// TIA Portal V16 export
// export: Created 2021-11-12T13:33:10.1366226Z, ExportSetting WithDefaults, DisplayName Totally Integrated Automation Portal, DisplayVersion V16 Update 3, DisplayName TIA Portal Version Control Interface, DisplayVersion V16 Update 2, DisplayName TIA Portal Openness, DisplayVersion V16 Update 3, DisplayName SINAMICS Startdrive Advanced, DisplayVersion V16 Update 5, DisplayName SINAMICS Startdrive G130, G150, S120, S150, SINAMICS MV, S210, DisplayVersion V16 Update 5, DisplayName SINAMICS Startdrive G110M, G120, G120C, G120D, G120P, G115D, DisplayVersion V16 Update 5, DisplayName STEP 7 Professional, DisplayVersion V16 Update 3, DisplayName STEP 7 Safety, DisplayVersion V16, DisplayName WinCC UA Professional, DisplayVersion V16 Update 3
FUNCTION_BLOCK "Station450"   // FB58, LAD
{ S7_Optimized_Access := 'TRUE' }
VERSION : 0.1
// stored: AutoNumber true, IsIECCheckEnabled false, IsRetainMemResEnabled false, MemoryReserve 100, SetENOAutomatically false, UDAEnableTagReadback false
   VAR
      SF_GL01_MA01 : "STD_Drive1";
      SF_GL02_MA01 { S7_SetPoint := 'True'} : "STD_Drive1";
      SF_GL03_MA01 { S7_SetPoint := 'True'} : "STD_Drive1";
      SF_GL04_MA01 { S7_SetPoint := 'True'} : "STD_Drive1";
      SF_UC21_TA1 { S7_SetPoint := 'True'} : "STD_Siemens_G120_CU240E_2_PN";
      SF_UC21_TA2 { S7_SetPoint := 'True'} : "STD_Siemens_G120_CU240E_2_PN";
      SF_UC21_TA3 { S7_SetPoint := 'True'} : "STD_Siemens_G120_CU240E_2_PN";
      SF_UC21_TA4 { S7_SetPoint := 'True'} : "STD_Siemens_G120_CU240E_2_PN";
      SF_BoxPartCounter { S7_SetPoint := 'True'} : "STD_PartCounter";
      SF_TON_BOX { S7_SetPoint := 'True'} : TON_TIME;
      SF_TOF_430TA01 { S7_SetPoint := 'True'} : TOF_TIME;   // TOF timer to stop conv after 430TA01 stopped
      SF_TOF_450TA01 { S7_SetPoint := 'True'} : TOF_TIME;   // TOF timer to stop conv after 450TA01 stopped
      SF_TOF_450TA02_1 { S7_SetPoint := 'True'} : TOF_TIME;   // TOF timer to stop conv after 450TA02 stopped
      SF_TOF_450TA02_2 { S7_SetPoint := 'True'} : TOF_TIME;   // TOF timer to stop conv after 450TA02 stopped
      SF_TOF_450TA04 { S7_SetPoint := 'True'} : TOF_TIME;   // TOF timer to stop conv after 450TA03 stopped
      SB1_PowerOk { S7_SetPoint := 'True'} : Bool;
      SB1BoxExchangeReq : Bool;   // Box - exchange request
      SF_CL01_Alarm { S7_SetPoint := 'True'} : "STD_DI_Mon";
      SF_CL01_Warning { S7_SetPoint := 'True'} : "STD_DI_Mon";
   END_VAR
   VAR_TEMP
      TS_GL01MA01 : "UDT_DriveControl";
      TS_GL02MA01 : "UDT_DriveControl";
      TS_GL03MA01 : "UDT_DriveControl";
      TS_GL04MA01 : "UDT_DriveControl";
      TS_UC21TA01 : Struct
         ReqDir1 : Bool;   // Move in direction 1
         ReqDir2 : Bool;   // Move in direction 2
         AckErr : Bool;   // Acknowledge error
         SpeedSP : Real;   // Speed setpoint
      END_STRUCT;
      TS_UC21TA02 : Struct
         ReqDir1 : Bool;   // Move in direction 1
         ReqDir2 : Bool;   // Move in direction 2
         AckErr : Bool;   // Acknowledge error
         SpeedSP : Real;   // Speed setpoint
      END_STRUCT;
      TS_UC21TA03 : Struct
         ReqDir1 : Bool;   // Move in direction 1
         ReqDir2 : Bool;   // Move in direction 2
         AckErr : Bool;   // Acknowledge error
         SpeedSP : Real;   // Speed setpoint
      END_STRUCT;
      TS_UC21TA04 : Struct
         ReqDir1 : Bool;   // Move in direction 1
         ReqDir2 : Bool;   // Move in direction 2
         AckErr : Bool;   // Acknowledge error
         SpeedSP : Real;   // Speed setpoint
      END_STRUCT;
      TI_NoOfParts : Int;   // Number of parts per one pulse
      TB1BoxFull : Bool;   // Box is full
   END_VAR
BEGIN

REGION Network 1: ***************ClearTemporary***************
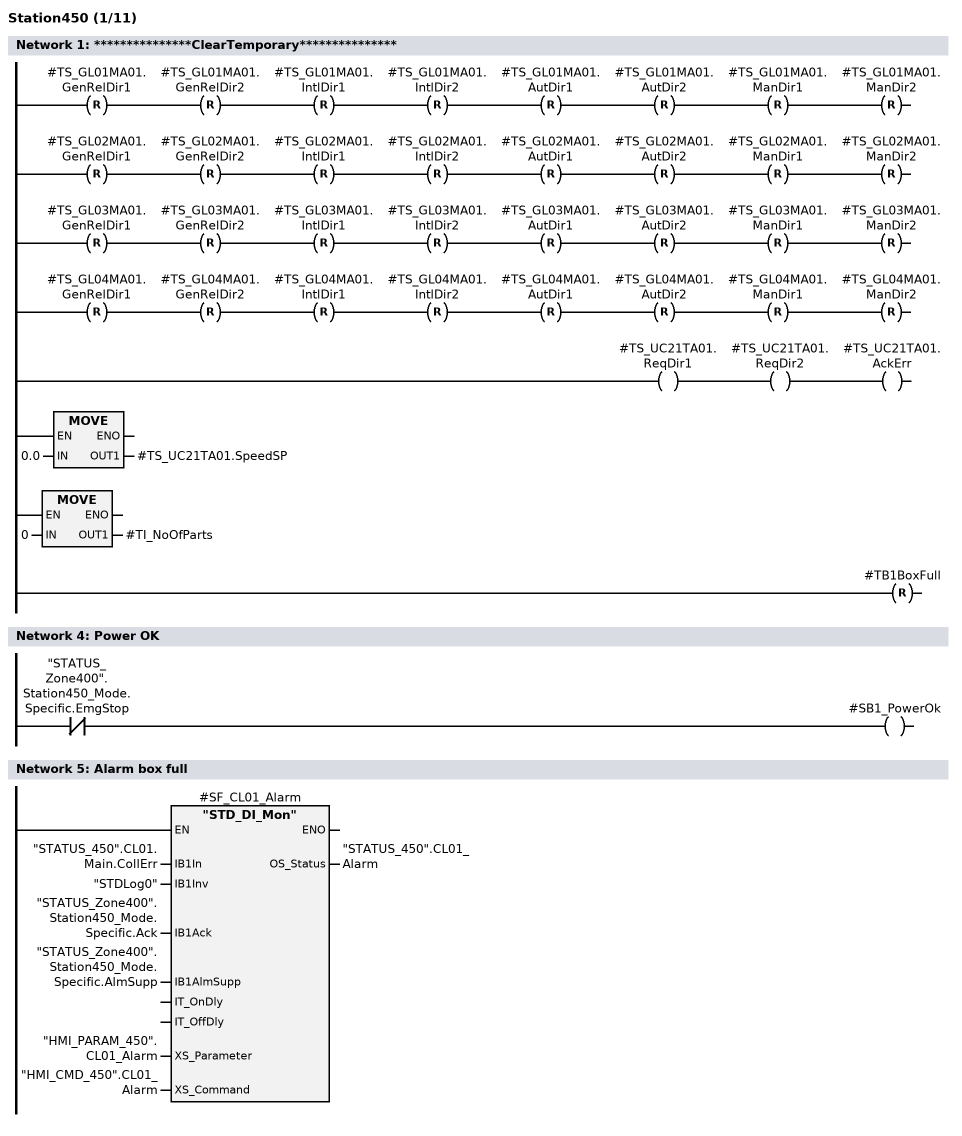
   RUNG wire#powerrail
      R_Coil( #TS_GL01MA01.GenRelDir1 )
      R_Coil( #TS_GL01MA01.GenRelDir2 )
      R_Coil( #TS_GL01MA01.IntlDir1 )
      R_Coil( #TS_GL01MA01.IntlDir2 )
      R_Coil( #TS_GL01MA01.AutDir1 )
      R_Coil( #TS_GL01MA01.AutDir2 )
      R_Coil( #TS_GL01MA01.ManDir1 )
      R_Coil( #TS_GL01MA01.ManDir2 )
   END_RUNG
   RUNG wire#powerrail
      R_Coil( #TS_GL02MA01.GenRelDir1 )
      R_Coil( #TS_GL02MA01.GenRelDir2 )
      R_Coil( #TS_GL02MA01.IntlDir1 )
      R_Coil( #TS_GL02MA01.IntlDir2 )
      R_Coil( #TS_GL02MA01.AutDir1 )
      R_Coil( #TS_GL02MA01.AutDir2 )
      R_Coil( #TS_GL02MA01.ManDir1 )
      R_Coil( #TS_GL02MA01.ManDir2 )
   END_RUNG
   RUNG wire#powerrail
      R_Coil( #TS_GL03MA01.GenRelDir1 )
      R_Coil( #TS_GL03MA01.GenRelDir2 )
      R_Coil( #TS_GL03MA01.IntlDir1 )
      R_Coil( #TS_GL03MA01.IntlDir2 )
      R_Coil( #TS_GL03MA01.AutDir1 )
      R_Coil( #TS_GL03MA01.AutDir2 )
      R_Coil( #TS_GL03MA01.ManDir1 )
      R_Coil( #TS_GL03MA01.ManDir2 )
   END_RUNG
   RUNG wire#powerrail
      R_Coil( #TS_GL04MA01.GenRelDir1 )
      R_Coil( #TS_GL04MA01.GenRelDir2 )
      R_Coil( #TS_GL04MA01.IntlDir1 )
      R_Coil( #TS_GL04MA01.IntlDir2 )
      R_Coil( #TS_GL04MA01.AutDir1 )
      R_Coil( #TS_GL04MA01.AutDir2 )
      R_Coil( #TS_GL04MA01.ManDir1 )
      R_Coil( #TS_GL04MA01.ManDir2 )
   END_RUNG
   RUNG wire#powerrail
      Coil( #TS_UC21TA01.ReqDir1 )
      Coil( #TS_UC21TA01.ReqDir2 )
      Coil( #TS_UC21TA01.AckErr )
   END_RUNG
   RUNG wire#powerrail
      Move(in := 0.0, out1 => #TS_UC21TA01.SpeedSP)
   END_RUNG
   RUNG wire#powerrail
      Move(in := 0, out1 => #TI_NoOfParts)
   END_RUNG
   RUNG wire#powerrail
      R_Coil( #TB1BoxFull )
   END_RUNG
   // the same network as SCL:
   #TS_GL01MA01.GenRelDir1 := FALSE;
   #TS_GL01MA01.GenRelDir2 := FALSE;
   #TS_GL01MA01.IntlDir1 := FALSE;
   #TS_GL01MA01.IntlDir2 := FALSE;
   #TS_GL01MA01.AutDir1 := FALSE;
   #TS_GL01MA01.AutDir2 := FALSE;
   #TS_GL01MA01.ManDir1 := FALSE;
   #TS_GL01MA01.ManDir2 := FALSE;
   #TS_GL02MA01.GenRelDir1 := FALSE;
   #TS_GL02MA01.GenRelDir2 := FALSE;
   #TS_GL02MA01.IntlDir1 := FALSE;
   #TS_GL02MA01.IntlDir2 := FALSE;
   #TS_GL02MA01.AutDir1 := FALSE;
   #TS_GL02MA01.AutDir2 := FALSE;
   #TS_GL02MA01.ManDir1 := FALSE;
   #TS_GL02MA01.ManDir2 := FALSE;
   #TS_GL03MA01.GenRelDir1 := FALSE;
   #TS_GL03MA01.GenRelDir2 := FALSE;
   #TS_GL03MA01.IntlDir1 := FALSE;
   #TS_GL03MA01.IntlDir2 := FALSE;
   #TS_GL03MA01.AutDir1 := FALSE;
   #TS_GL03MA01.AutDir2 := FALSE;
   #TS_GL03MA01.ManDir1 := FALSE;
   #TS_GL03MA01.ManDir2 := FALSE;
   #TS_GL04MA01.GenRelDir1 := FALSE;
   #TS_GL04MA01.GenRelDir2 := FALSE;
   #TS_GL04MA01.IntlDir1 := FALSE;
   #TS_GL04MA01.IntlDir2 := FALSE;
   #TS_GL04MA01.AutDir1 := FALSE;
   #TS_GL04MA01.AutDir2 := FALSE;
   #TS_GL04MA01.ManDir1 := FALSE;
   #TS_GL04MA01.ManDir2 := FALSE;
   #TS_UC21TA01.ReqDir1 := TRUE;
   #TS_UC21TA01.ReqDir2 := TRUE;
   #TS_UC21TA01.AckErr := TRUE;
   #TS_UC21TA01.SpeedSP := 0.0;
   #TI_NoOfParts := 0;
   #TB1BoxFull := FALSE;
END_REGION

REGION Network 2: ***************SensorsAlarms***************
END_REGION

REGION Network 3: ***************ProcesAlarms***************
END_REGION

REGION Network 4: Power OK
   RUNG wire#powerrail
      I_Contact( "STATUS_Zone400".Station450_Mode.Specific.EmgStop )
      Coil( #SB1_PowerOk )
   END_RUNG
   // the same network as SCL:
   #SB1_PowerOk := NOT "STATUS_Zone400".Station450_Mode.Specific.EmgStop;
END_REGION

REGION Network 5: Alarm box full
   RUNG wire#powerrail
      #SF_CL01_Alarm(IB1In := "STATUS_450".CL01.Main.CollErr, IB1Inv := "STDLog0", IB1Ack := "STATUS_Zone400".Station450_Mode.Specific.Ack, IB1AlmSupp := "STATUS_Zone400".Station450_Mode.Specific.AlmSupp, IT_OnDly :=, IT_OffDly :=, XS_Parameter := "HMI_PARAM_450".CL01_Alarm, XS_Command := "HMI_CMD_450".CL01_Alarm, OS_Status => "STATUS_450".CL01_Alarm)
   END_RUNG
   // the same network as SCL:
   #SF_CL01_Alarm(IB1In := "STATUS_450".CL01.Main.CollErr,   // "STD_DI_Mon"
                  IB1Inv := "STDLog0",
                  IB1Ack := "STATUS_Zone400".Station450_Mode.Specific.Ack,
                  IB1AlmSupp := "STATUS_Zone400".Station450_Mode.Specific.AlmSupp,
                  XS_Parameter := "HMI_PARAM_450".CL01_Alarm,
                  XS_Command := "HMI_CMD_450".CL01_Alarm,
                  OS_Status => "STATUS_450".CL01_Alarm);
END_REGION

REGION Network 6: Warning box almost full
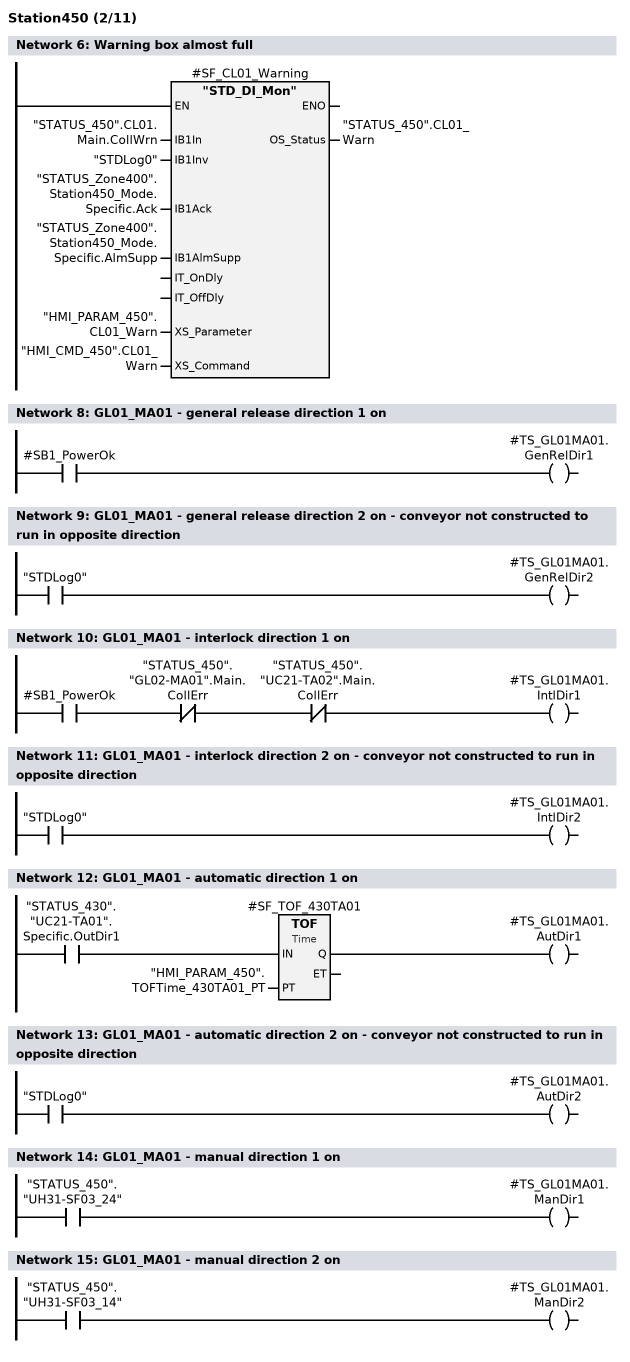
   RUNG wire#powerrail
      #SF_CL01_Warning(IB1In := "STATUS_450".CL01.Main.CollWrn, IB1Inv := "STDLog0", IB1Ack := "STATUS_Zone400".Station450_Mode.Specific.Ack, IB1AlmSupp := "STATUS_Zone400".Station450_Mode.Specific.AlmSupp, IT_OnDly :=, IT_OffDly :=, XS_Parameter := "HMI_PARAM_450".CL01_Warn, XS_Command := "HMI_CMD_450".CL01_Warn, OS_Status => "STATUS_450".CL01_Warn)
   END_RUNG
   // the same network as SCL:
   #SF_CL01_Warning(IB1In := "STATUS_450".CL01.Main.CollWrn,   // "STD_DI_Mon"
                    IB1Inv := "STDLog0",
                    IB1Ack := "STATUS_Zone400".Station450_Mode.Specific.Ack,
                    IB1AlmSupp := "STATUS_Zone400".Station450_Mode.Specific.AlmSupp,
                    XS_Parameter := "HMI_PARAM_450".CL01_Warn,
                    XS_Command := "HMI_CMD_450".CL01_Warn,
                    OS_Status => "STATUS_450".CL01_Warn);
END_REGION

REGION Network 7: ***************GL01_MA01 Conveyor M2***************
END_REGION

REGION Network 8: GL01_MA01 - general release direction 1 on
   RUNG wire#powerrail
      Contact( #SB1_PowerOk )
      Coil( #TS_GL01MA01.GenRelDir1 )
   END_RUNG
   // the same network as SCL:
   #TS_GL01MA01.GenRelDir1 := #SB1_PowerOk;
END_REGION

REGION Network 9: GL01_MA01 - general release direction 2 on - conveyor not constructed to run in opposite direction
   RUNG wire#powerrail
      Contact( "STDLog0" )
      Coil( #TS_GL01MA01.GenRelDir2 )
   END_RUNG
   // the same network as SCL:
   #TS_GL01MA01.GenRelDir2 := "STDLog0";
END_REGION

REGION Network 10: GL01_MA01 - interlock direction 1 on
   RUNG wire#powerrail
      Contact( #SB1_PowerOk )
      I_Contact( "STATUS_450"."GL02-MA01".Main.CollErr )
      I_Contact( "STATUS_450"."UC21-TA02".Main.CollErr )
      Coil( #TS_GL01MA01.IntlDir1 )
   END_RUNG
   // the same network as SCL:
   #TS_GL01MA01.IntlDir1 := #SB1_PowerOk AND NOT "STATUS_450"."GL02-MA01".Main.CollErr AND NOT "STATUS_450"."UC21-TA02".Main.CollErr;
END_REGION

REGION Network 11: GL01_MA01 - interlock direction 2 on - conveyor not constructed to run in opposite direction
   RUNG wire#powerrail
      Contact( "STDLog0" )
      Coil( #TS_GL01MA01.IntlDir2 )
   END_RUNG
   // the same network as SCL:
   #TS_GL01MA01.IntlDir2 := "STDLog0";
END_REGION

REGION Network 12: GL01_MA01 - automatic direction 1 on
   RUNG wire#powerrail
      Contact( "STATUS_430"."UC21-TA01".Specific.OutDir1 )
      { S7_Templates := "time_type := Time" } #SF_TOF_430TA01.TOF(pt := "HMI_PARAM_450".TOFTime_430TA01_PT, et =>)
      Coil( #TS_GL01MA01.AutDir1 )
   END_RUNG
   // the same network as SCL:
   #SF_TOF_430TA01(IN := "STATUS_430"."UC21-TA01".Specific.OutDir1, PT := "HMI_PARAM_450".TOFTime_430TA01_PT);   // TOF
   #TS_GL01MA01.AutDir1 := #SF_TOF_430TA01.Q;
END_REGION

REGION Network 13: GL01_MA01 - automatic direction 2 on - conveyor not constructed to run in opposite direction
   RUNG wire#powerrail
      Contact( "STDLog0" )
      Coil( #TS_GL01MA01.AutDir2 )
   END_RUNG
   // the same network as SCL:
   #TS_GL01MA01.AutDir2 := "STDLog0";
END_REGION

REGION Network 14: GL01_MA01 - manual direction 1 on
   RUNG wire#powerrail
      Contact( "STATUS_450"."UH31-SF03_24" )
      Coil( #TS_GL01MA01.ManDir1 )
   END_RUNG
   // the same network as SCL:
   #TS_GL01MA01.ManDir1 := "STATUS_450"."UH31-SF03_24";
END_REGION

REGION Network 15: GL01_MA01 - manual direction 2 on
   RUNG wire#powerrail
      Contact( "STATUS_450"."UH31-SF03_14" )
      Coil( #TS_GL01MA01.ManDir2 )
   END_RUNG
   // the same network as SCL:
   #TS_GL01MA01.ManDir2 := "STATUS_450"."UH31-SF03_14";
END_REGION

REGION Network 16: GL01_MA01 Drive block call
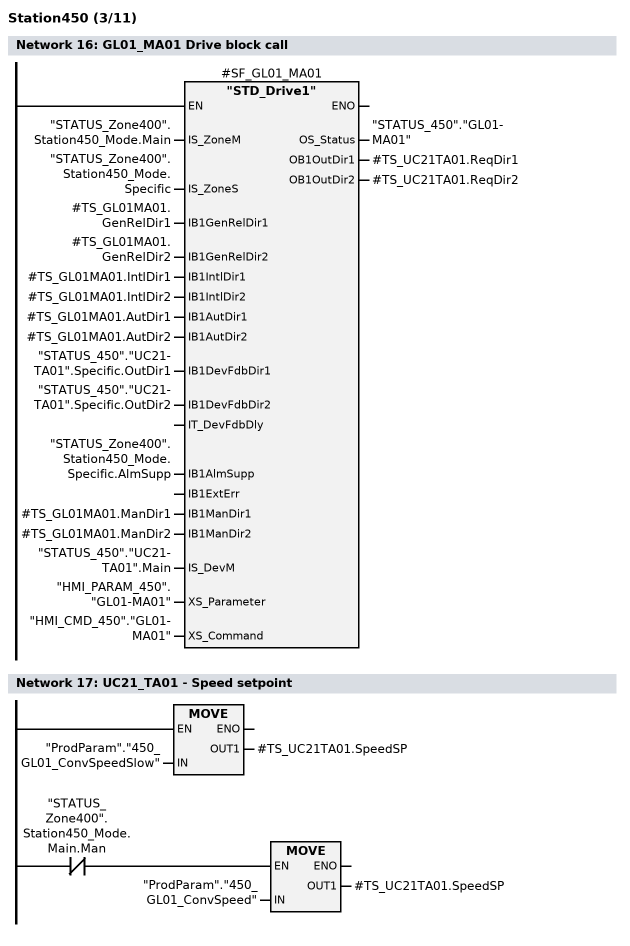
   RUNG wire#powerrail
      #SF_GL01_MA01(IS_ZoneM := "STATUS_Zone400".Station450_Mode.Main, IS_ZoneS := "STATUS_Zone400".Station450_Mode.Specific, IB1GenRelDir1 := #TS_GL01MA01.GenRelDir1, IB1GenRelDir2 := #TS_GL01MA01.GenRelDir2, IB1IntlDir1 := #TS_GL01MA01.IntlDir1, IB1IntlDir2 := #TS_GL01MA01.IntlDir2, IB1AutDir1 := #TS_GL01MA01.AutDir1, IB1AutDir2 := #TS_GL01MA01.AutDir2, IB1DevFdbDir1 := "STATUS_450"."UC21-TA01".Specific.OutDir1, IB1DevFdbDir2 := "STATUS_450"."UC21-TA01".Specific.OutDir2, IT_DevFdbDly :=, IB1AlmSupp := "STATUS_Zone400".Station450_Mode.Specific.AlmSupp, IB1ExtErr :=, IB1ManDir1 := #TS_GL01MA01.ManDir1, IB1ManDir2 := #TS_GL01MA01.ManDir2, IS_DevM := "STATUS_450"."UC21-TA01".Main, XS_Parameter := "HMI_PARAM_450"."GL01-MA01", XS_Command := "HMI_CMD_450"."GL01-MA01", OS_Status => "STATUS_450"."GL01-MA01", OB1OutDir1 => #TS_UC21TA01.ReqDir1, OB1OutDir2 => #TS_UC21TA01.ReqDir2)
   END_RUNG
   // the same network as SCL:
   #SF_GL01_MA01(IS_ZoneM := "STATUS_Zone400".Station450_Mode.Main,   // "STD_Drive1"
                 IS_ZoneS := "STATUS_Zone400".Station450_Mode.Specific,
                 IB1GenRelDir1 := #TS_GL01MA01.GenRelDir1,
                 IB1GenRelDir2 := #TS_GL01MA01.GenRelDir2,
                 IB1IntlDir1 := #TS_GL01MA01.IntlDir1,
                 IB1IntlDir2 := #TS_GL01MA01.IntlDir2,
                 IB1AutDir1 := #TS_GL01MA01.AutDir1,
                 IB1AutDir2 := #TS_GL01MA01.AutDir2,
                 IB1DevFdbDir1 := "STATUS_450"."UC21-TA01".Specific.OutDir1,
                 IB1DevFdbDir2 := "STATUS_450"."UC21-TA01".Specific.OutDir2,
                 IB1AlmSupp := "STATUS_Zone400".Station450_Mode.Specific.AlmSupp,
                 IB1ManDir1 := #TS_GL01MA01.ManDir1,
                 IB1ManDir2 := #TS_GL01MA01.ManDir2,
                 IS_DevM := "STATUS_450"."UC21-TA01".Main,
                 XS_Parameter := "HMI_PARAM_450"."GL01-MA01",
                 XS_Command := "HMI_CMD_450"."GL01-MA01",
                 OS_Status => "STATUS_450"."GL01-MA01",
                 OB1OutDir1 => #TS_UC21TA01.ReqDir1,
                 OB1OutDir2 => #TS_UC21TA01.ReqDir2);
END_REGION

REGION Network 17: UC21_TA01 - Speed setpoint
   RUNG wire#powerrail
      Move(in := "ProdParam"."450_GL01_ConvSpeedSlow", out1 => #TS_UC21TA01.SpeedSP)
   END_RUNG
   RUNG wire#powerrail
      I_Contact( "STATUS_Zone400".Station450_Mode.Main.Man )
      Move(in := "ProdParam"."450_GL01_ConvSpeed", out1 => #TS_UC21TA01.SpeedSP)
   END_RUNG
   // the same network as SCL:
   #TS_UC21TA01.SpeedSP := "ProdParam"."450_GL01_ConvSpeedSlow";
   IF NOT "STATUS_Zone400".Station450_Mode.Main.Man THEN
       #TS_UC21TA01.SpeedSP := "ProdParam"."450_GL01_ConvSpeed";
   END_IF;
END_REGION

REGION Network 18: UC21_TA01 - Frequency convertor block call
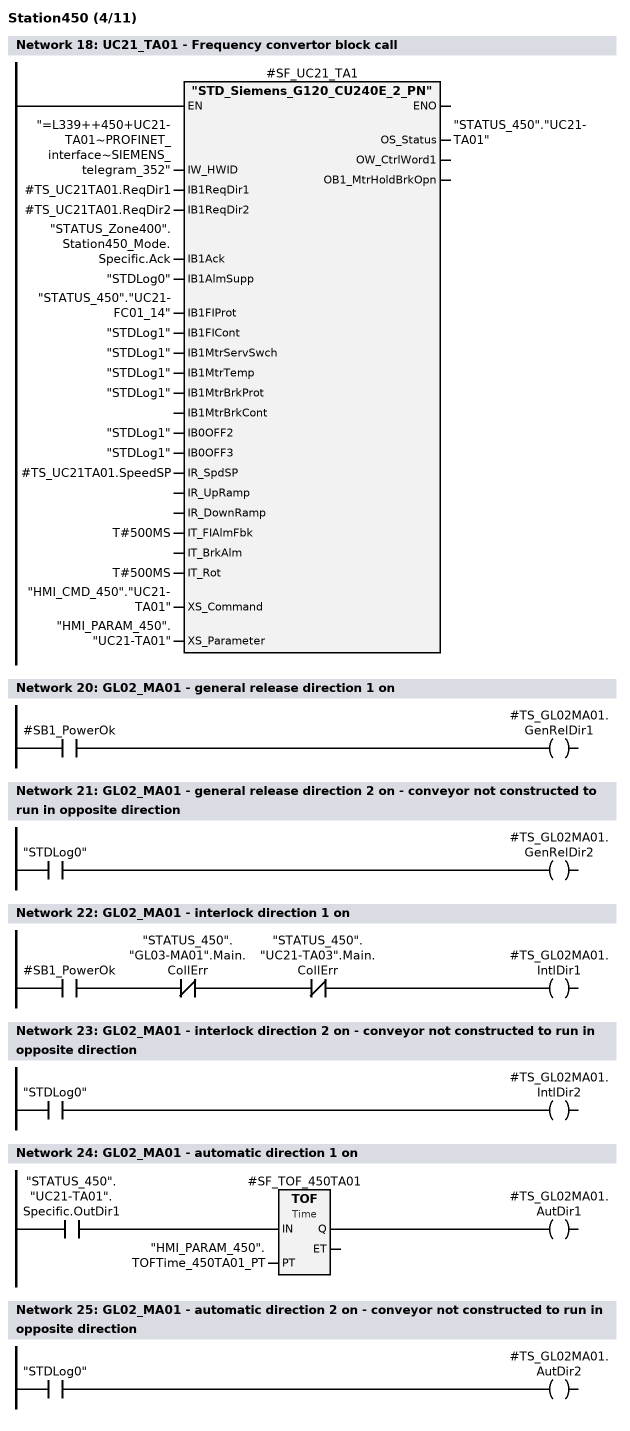
   RUNG wire#powerrail
      #SF_UC21_TA1(IW_HWID := "=L339++450+UC21-TA01~PROFINET_interface~SIEMENS_telegram_352", IB1ReqDir1 := #TS_UC21TA01.ReqDir1, IB1ReqDir2 := #TS_UC21TA01.ReqDir2, IB1Ack := "STATUS_Zone400".Station450_Mode.Specific.Ack, IB1AlmSupp := "STDLog0", IB1FIProt := "STATUS_450"."UC21-FC01_14", IB1FICont := "STDLog1", IB1MtrServSwch := "STDLog1", IB1MtrTemp := "STDLog1", IB1MtrBrkProt := "STDLog1", IB1MtrBrkCont :=, IB0OFF2 := "STDLog1", IB0OFF3 := "STDLog1", IR_SpdSP := #TS_UC21TA01.SpeedSP, IR_UpRamp :=, IR_DownRamp :=, IT_FIAlmFbk := T#500MS, IT_BrkAlm :=, IT_Rot := T#500MS, XS_Command := "HMI_CMD_450"."UC21-TA01", XS_Parameter := "HMI_PARAM_450"."UC21-TA01", OS_Status => "STATUS_450"."UC21-TA01", OW_CtrlWord1 =>, OB1_MtrHoldBrkOpn =>)
   END_RUNG
   // the same network as SCL:
   #SF_UC21_TA1(IW_HWID := "=L339++450+UC21-TA01~PROFINET_interface~SIEMENS_telegram_352",   // "STD_Siemens_G120_CU240E_2_PN"
                IB1ReqDir1 := #TS_UC21TA01.ReqDir1,
                IB1ReqDir2 := #TS_UC21TA01.ReqDir2,
                IB1Ack := "STATUS_Zone400".Station450_Mode.Specific.Ack,
                IB1AlmSupp := "STDLog0",
                IB1FIProt := "STATUS_450"."UC21-FC01_14",
                IB1FICont := "STDLog1",
                IB1MtrServSwch := "STDLog1",
                IB1MtrTemp := "STDLog1",
                IB1MtrBrkProt := "STDLog1",
                IB0OFF2 := "STDLog1",
                IB0OFF3 := "STDLog1",
                IR_SpdSP := #TS_UC21TA01.SpeedSP,
                IT_FIAlmFbk := T#500MS,
                IT_Rot := T#500MS,
                XS_Command := "HMI_CMD_450"."UC21-TA01",
                XS_Parameter := "HMI_PARAM_450"."UC21-TA01",
                OS_Status => "STATUS_450"."UC21-TA01");
END_REGION

REGION Network 19: ***************GL02_MA01 Conveyor M4***************
END_REGION

REGION Network 20: GL02_MA01 - general release direction 1 on
   RUNG wire#powerrail
      Contact( #SB1_PowerOk )
      Coil( #TS_GL02MA01.GenRelDir1 )
   END_RUNG
   // the same network as SCL:
   #TS_GL02MA01.GenRelDir1 := #SB1_PowerOk;
END_REGION

REGION Network 21: GL02_MA01 - general release direction 2 on - conveyor not constructed to run in opposite direction
   RUNG wire#powerrail
      Contact( "STDLog0" )
      Coil( #TS_GL02MA01.GenRelDir2 )
   END_RUNG
   // the same network as SCL:
   #TS_GL02MA01.GenRelDir2 := "STDLog0";
END_REGION

REGION Network 22: GL02_MA01 - interlock direction 1 on
   RUNG wire#powerrail
      Contact( #SB1_PowerOk )
      I_Contact( "STATUS_450"."GL03-MA01".Main.CollErr )
      I_Contact( "STATUS_450"."UC21-TA03".Main.CollErr )
      Coil( #TS_GL02MA01.IntlDir1 )
   END_RUNG
   // the same network as SCL:
   #TS_GL02MA01.IntlDir1 := #SB1_PowerOk AND NOT "STATUS_450"."GL03-MA01".Main.CollErr AND NOT "STATUS_450"."UC21-TA03".Main.CollErr;
END_REGION

REGION Network 23: GL02_MA01 - interlock direction 2 on - conveyor not constructed to run in opposite direction
   RUNG wire#powerrail
      Contact( "STDLog0" )
      Coil( #TS_GL02MA01.IntlDir2 )
   END_RUNG
   // the same network as SCL:
   #TS_GL02MA01.IntlDir2 := "STDLog0";
END_REGION

REGION Network 24: GL02_MA01 - automatic direction 1 on
   RUNG wire#powerrail
      Contact( "STATUS_450"."UC21-TA01".Specific.OutDir1 )
      { S7_Templates := "time_type := Time" } #SF_TOF_450TA01.TOF(pt := "HMI_PARAM_450".TOFTime_450TA01_PT, et =>)
      Coil( #TS_GL02MA01.AutDir1 )
   END_RUNG
   // the same network as SCL:
   #SF_TOF_450TA01(IN := "STATUS_450"."UC21-TA01".Specific.OutDir1, PT := "HMI_PARAM_450".TOFTime_450TA01_PT);   // TOF
   #TS_GL02MA01.AutDir1 := #SF_TOF_450TA01.Q;
END_REGION

REGION Network 25: GL02_MA01 - automatic direction 2 on - conveyor not constructed to run in opposite direction
   RUNG wire#powerrail
      Contact( "STDLog0" )
      Coil( #TS_GL02MA01.AutDir2 )
   END_RUNG
   // the same network as SCL:
   #TS_GL02MA01.AutDir2 := "STDLog0";
END_REGION

REGION Network 26: GL02_MA01 - manual direction 1 on
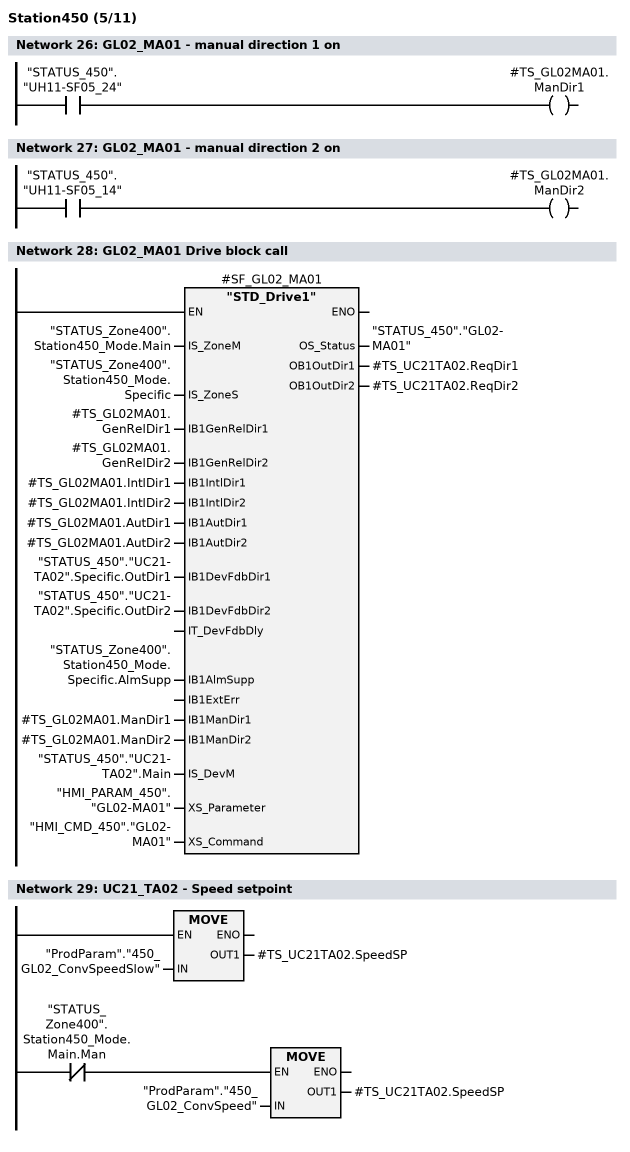
   RUNG wire#powerrail
      Contact( "STATUS_450"."UH11-SF05_24" )
      Coil( #TS_GL02MA01.ManDir1 )
   END_RUNG
   // the same network as SCL:
   #TS_GL02MA01.ManDir1 := "STATUS_450"."UH11-SF05_24";
END_REGION

REGION Network 27: GL02_MA01 - manual direction 2 on
   RUNG wire#powerrail
      Contact( "STATUS_450"."UH11-SF05_14" )
      Coil( #TS_GL02MA01.ManDir2 )
   END_RUNG
   // the same network as SCL:
   #TS_GL02MA01.ManDir2 := "STATUS_450"."UH11-SF05_14";
END_REGION

REGION Network 28: GL02_MA01 Drive block call
   RUNG wire#powerrail
      #SF_GL02_MA01(IS_ZoneM := "STATUS_Zone400".Station450_Mode.Main, IS_ZoneS := "STATUS_Zone400".Station450_Mode.Specific, IB1GenRelDir1 := #TS_GL02MA01.GenRelDir1, IB1GenRelDir2 := #TS_GL02MA01.GenRelDir2, IB1IntlDir1 := #TS_GL02MA01.IntlDir1, IB1IntlDir2 := #TS_GL02MA01.IntlDir2, IB1AutDir1 := #TS_GL02MA01.AutDir1, IB1AutDir2 := #TS_GL02MA01.AutDir2, IB1DevFdbDir1 := "STATUS_450"."UC21-TA02".Specific.OutDir1, IB1DevFdbDir2 := "STATUS_450"."UC21-TA02".Specific.OutDir2, IT_DevFdbDly :=, IB1AlmSupp := "STATUS_Zone400".Station450_Mode.Specific.AlmSupp, IB1ExtErr :=, IB1ManDir1 := #TS_GL02MA01.ManDir1, IB1ManDir2 := #TS_GL02MA01.ManDir2, IS_DevM := "STATUS_450"."UC21-TA02".Main, XS_Parameter := "HMI_PARAM_450"."GL02-MA01", XS_Command := "HMI_CMD_450"."GL02-MA01", OS_Status => "STATUS_450"."GL02-MA01", OB1OutDir1 => #TS_UC21TA02.ReqDir1, OB1OutDir2 => #TS_UC21TA02.ReqDir2)
   END_RUNG
   // the same network as SCL:
   #SF_GL02_MA01(IS_ZoneM := "STATUS_Zone400".Station450_Mode.Main,   // "STD_Drive1"
                 IS_ZoneS := "STATUS_Zone400".Station450_Mode.Specific,
                 IB1GenRelDir1 := #TS_GL02MA01.GenRelDir1,
                 IB1GenRelDir2 := #TS_GL02MA01.GenRelDir2,
                 IB1IntlDir1 := #TS_GL02MA01.IntlDir1,
                 IB1IntlDir2 := #TS_GL02MA01.IntlDir2,
                 IB1AutDir1 := #TS_GL02MA01.AutDir1,
                 IB1AutDir2 := #TS_GL02MA01.AutDir2,
                 IB1DevFdbDir1 := "STATUS_450"."UC21-TA02".Specific.OutDir1,
                 IB1DevFdbDir2 := "STATUS_450"."UC21-TA02".Specific.OutDir2,
                 IB1AlmSupp := "STATUS_Zone400".Station450_Mode.Specific.AlmSupp,
                 IB1ManDir1 := #TS_GL02MA01.ManDir1,
                 IB1ManDir2 := #TS_GL02MA01.ManDir2,
                 IS_DevM := "STATUS_450"."UC21-TA02".Main,
                 XS_Parameter := "HMI_PARAM_450"."GL02-MA01",
                 XS_Command := "HMI_CMD_450"."GL02-MA01",
                 OS_Status => "STATUS_450"."GL02-MA01",
                 OB1OutDir1 => #TS_UC21TA02.ReqDir1,
                 OB1OutDir2 => #TS_UC21TA02.ReqDir2);
END_REGION

REGION Network 29: UC21_TA02 - Speed setpoint
   RUNG wire#powerrail
      Move(in := "ProdParam"."450_GL02_ConvSpeedSlow", out1 => #TS_UC21TA02.SpeedSP)
   END_RUNG
   RUNG wire#powerrail
      I_Contact( "STATUS_Zone400".Station450_Mode.Main.Man )
      Move(in := "ProdParam"."450_GL02_ConvSpeed", out1 => #TS_UC21TA02.SpeedSP)
   END_RUNG
   // the same network as SCL:
   #TS_UC21TA02.SpeedSP := "ProdParam"."450_GL02_ConvSpeedSlow";
   IF NOT "STATUS_Zone400".Station450_Mode.Main.Man THEN
       #TS_UC21TA02.SpeedSP := "ProdParam"."450_GL02_ConvSpeed";
   END_IF;
END_REGION

REGION Network 30: UC21_TA02 - Frequency convertor block call
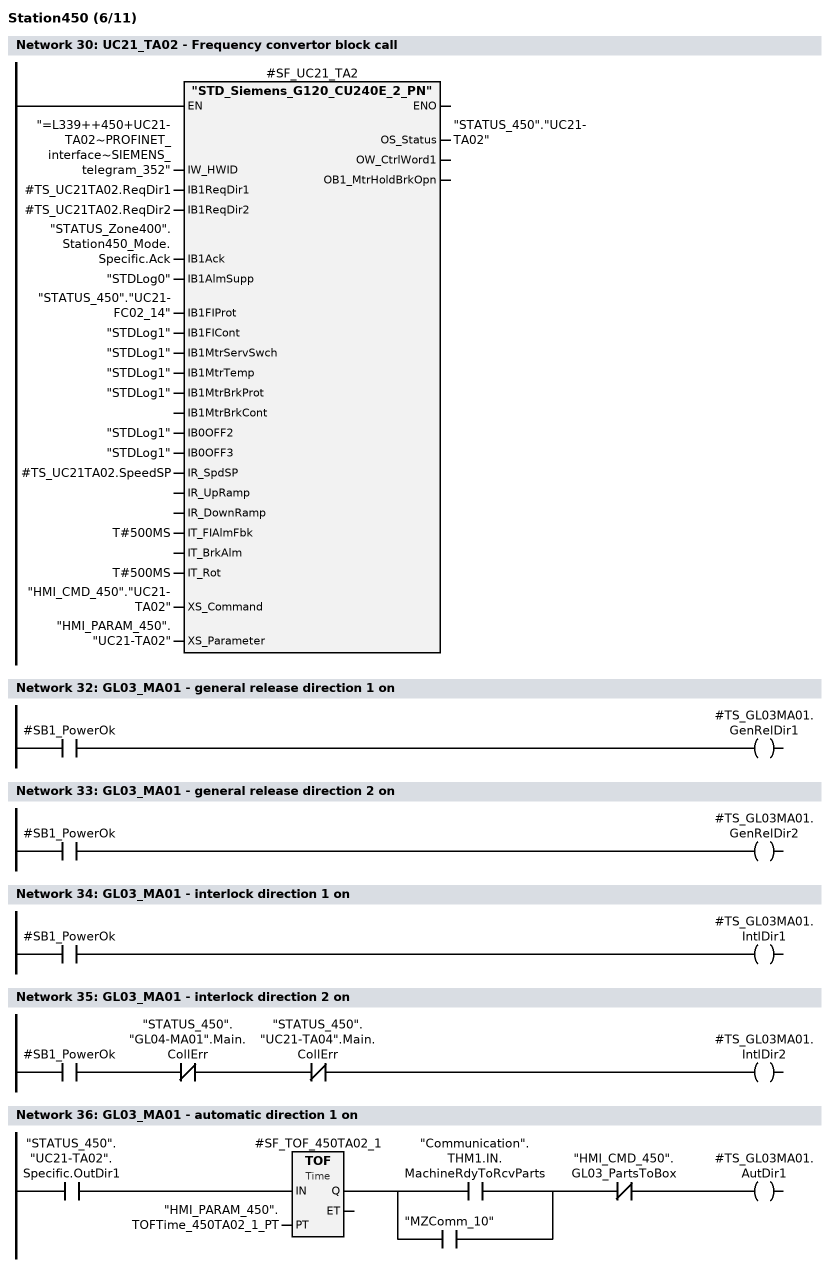
   RUNG wire#powerrail
      #SF_UC21_TA2(IW_HWID := "=L339++450+UC21-TA02~PROFINET_interface~SIEMENS_telegram_352", IB1ReqDir1 := #TS_UC21TA02.ReqDir1, IB1ReqDir2 := #TS_UC21TA02.ReqDir2, IB1Ack := "STATUS_Zone400".Station450_Mode.Specific.Ack, IB1AlmSupp := "STDLog0", IB1FIProt := "STATUS_450"."UC21-FC02_14", IB1FICont := "STDLog1", IB1MtrServSwch := "STDLog1", IB1MtrTemp := "STDLog1", IB1MtrBrkProt := "STDLog1", IB1MtrBrkCont :=, IB0OFF2 := "STDLog1", IB0OFF3 := "STDLog1", IR_SpdSP := #TS_UC21TA02.SpeedSP, IR_UpRamp :=, IR_DownRamp :=, IT_FIAlmFbk := T#500MS, IT_BrkAlm :=, IT_Rot := T#500MS, XS_Command := "HMI_CMD_450"."UC21-TA02", XS_Parameter := "HMI_PARAM_450"."UC21-TA02", OS_Status => "STATUS_450"."UC21-TA02", OW_CtrlWord1 =>, OB1_MtrHoldBrkOpn =>)
   END_RUNG
   // the same network as SCL:
   #SF_UC21_TA2(IW_HWID := "=L339++450+UC21-TA02~PROFINET_interface~SIEMENS_telegram_352",   // "STD_Siemens_G120_CU240E_2_PN"
                IB1ReqDir1 := #TS_UC21TA02.ReqDir1,
                IB1ReqDir2 := #TS_UC21TA02.ReqDir2,
                IB1Ack := "STATUS_Zone400".Station450_Mode.Specific.Ack,
                IB1AlmSupp := "STDLog0",
                IB1FIProt := "STATUS_450"."UC21-FC02_14",
                IB1FICont := "STDLog1",
                IB1MtrServSwch := "STDLog1",
                IB1MtrTemp := "STDLog1",
                IB1MtrBrkProt := "STDLog1",
                IB0OFF2 := "STDLog1",
                IB0OFF3 := "STDLog1",
                IR_SpdSP := #TS_UC21TA02.SpeedSP,
                IT_FIAlmFbk := T#500MS,
                IT_Rot := T#500MS,
                XS_Command := "HMI_CMD_450"."UC21-TA02",
                XS_Parameter := "HMI_PARAM_450"."UC21-TA02",
                OS_Status => "STATUS_450"."UC21-TA02");
END_REGION

REGION Network 31: ***************GL03_MA01 Conveyor M7.1***************
END_REGION

REGION Network 32: GL03_MA01 - general release direction 1 on
   RUNG wire#powerrail
      Contact( #SB1_PowerOk )
      Coil( #TS_GL03MA01.GenRelDir1 )
   END_RUNG
   // the same network as SCL:
   #TS_GL03MA01.GenRelDir1 := #SB1_PowerOk;
END_REGION

REGION Network 33: GL03_MA01 - general release direction 2 on
   RUNG wire#powerrail
      Contact( #SB1_PowerOk )
      Coil( #TS_GL03MA01.GenRelDir2 )
   END_RUNG
   // the same network as SCL:
   #TS_GL03MA01.GenRelDir2 := #SB1_PowerOk;
END_REGION

REGION Network 34: GL03_MA01 - interlock direction 1 on
   RUNG wire#powerrail
      Contact( #SB1_PowerOk )
      Coil( #TS_GL03MA01.IntlDir1 )
   END_RUNG
   // the same network as SCL:
   #TS_GL03MA01.IntlDir1 := #SB1_PowerOk;
END_REGION

REGION Network 35: GL03_MA01 - interlock direction 2 on
   RUNG wire#powerrail
      Contact( #SB1_PowerOk )
      I_Contact( "STATUS_450"."GL04-MA01".Main.CollErr )
      I_Contact( "STATUS_450"."UC21-TA04".Main.CollErr )
      Coil( #TS_GL03MA01.IntlDir2 )
   END_RUNG
   // the same network as SCL:
   #TS_GL03MA01.IntlDir2 := #SB1_PowerOk AND NOT "STATUS_450"."GL04-MA01".Main.CollErr AND NOT "STATUS_450"."UC21-TA04".Main.CollErr;
END_REGION

REGION Network 36: GL03_MA01 - automatic direction 1 on
   RUNG wire#powerrail
      Contact( "STATUS_450"."UC21-TA02".Specific.OutDir1 )
      { S7_Templates := "time_type := Time" } #SF_TOF_450TA02_1.TOF(pt := "HMI_PARAM_450".TOFTime_450TA02_1_PT, et =>)
      wire#w1
      Contact( "Communication".THM1.IN.MachineRdyToRcvParts )
      wire#w2
      I_Contact( "HMI_CMD_450".GL03_PartsToBox )
      Coil( #TS_GL03MA01.AutDir1 )
   END_RUNG
   RUNG wire#w1
      Contact( "MZComm_10" )
   END_RUNG wire#w2
   // the same network as SCL:
   #SF_TOF_450TA02_1(IN := "STATUS_450"."UC21-TA02".Specific.OutDir1,   // TOF
                     PT := "HMI_PARAM_450".TOFTime_450TA02_1_PT);
   #TS_GL03MA01.AutDir1 := #SF_TOF_450TA02_1.Q AND ("Communication".THM1.IN.MachineRdyToRcvParts OR "MZComm_10") AND NOT "HMI_CMD_450".GL03_PartsToBox;
END_REGION

REGION Network 37: GL03_MA01 - automatic direction 2 on
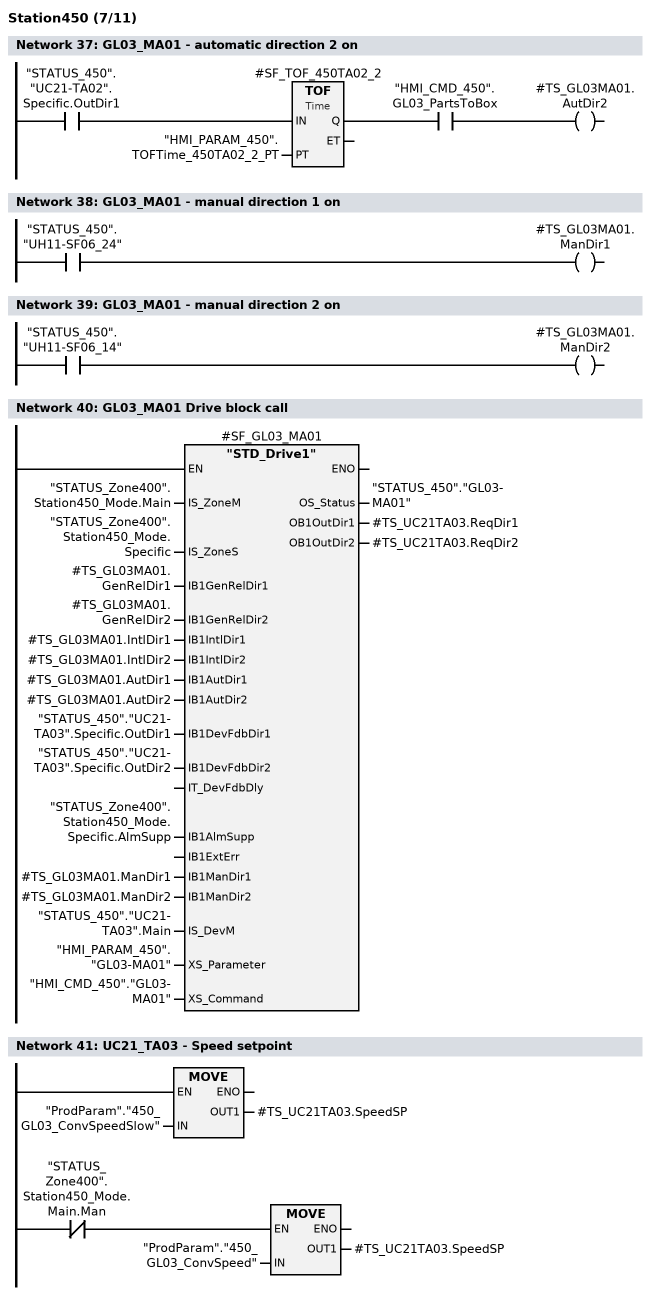
   RUNG wire#powerrail
      Contact( "STATUS_450"."UC21-TA02".Specific.OutDir1 )
      { S7_Templates := "time_type := Time" } #SF_TOF_450TA02_2.TOF(pt := "HMI_PARAM_450".TOFTime_450TA02_2_PT, et =>)
      Contact( "HMI_CMD_450".GL03_PartsToBox )
      Coil( #TS_GL03MA01.AutDir2 )
   END_RUNG
   // the same network as SCL:
   #SF_TOF_450TA02_2(IN := "STATUS_450"."UC21-TA02".Specific.OutDir1,   // TOF
                     PT := "HMI_PARAM_450".TOFTime_450TA02_2_PT);
   #TS_GL03MA01.AutDir2 := #SF_TOF_450TA02_2.Q AND "HMI_CMD_450".GL03_PartsToBox;
END_REGION

REGION Network 38: GL03_MA01 - manual direction 1 on
   RUNG wire#powerrail
      Contact( "STATUS_450"."UH11-SF06_24" )
      Coil( #TS_GL03MA01.ManDir1 )
   END_RUNG
   // the same network as SCL:
   #TS_GL03MA01.ManDir1 := "STATUS_450"."UH11-SF06_24";
END_REGION

REGION Network 39: GL03_MA01 - manual direction 2 on
   RUNG wire#powerrail
      Contact( "STATUS_450"."UH11-SF06_14" )
      Coil( #TS_GL03MA01.ManDir2 )
   END_RUNG
   // the same network as SCL:
   #TS_GL03MA01.ManDir2 := "STATUS_450"."UH11-SF06_14";
END_REGION

REGION Network 40: GL03_MA01 Drive block call
   RUNG wire#powerrail
      #SF_GL03_MA01(IS_ZoneM := "STATUS_Zone400".Station450_Mode.Main, IS_ZoneS := "STATUS_Zone400".Station450_Mode.Specific, IB1GenRelDir1 := #TS_GL03MA01.GenRelDir1, IB1GenRelDir2 := #TS_GL03MA01.GenRelDir2, IB1IntlDir1 := #TS_GL03MA01.IntlDir1, IB1IntlDir2 := #TS_GL03MA01.IntlDir2, IB1AutDir1 := #TS_GL03MA01.AutDir1, IB1AutDir2 := #TS_GL03MA01.AutDir2, IB1DevFdbDir1 := "STATUS_450"."UC21-TA03".Specific.OutDir1, IB1DevFdbDir2 := "STATUS_450"."UC21-TA03".Specific.OutDir2, IT_DevFdbDly :=, IB1AlmSupp := "STATUS_Zone400".Station450_Mode.Specific.AlmSupp, IB1ExtErr :=, IB1ManDir1 := #TS_GL03MA01.ManDir1, IB1ManDir2 := #TS_GL03MA01.ManDir2, IS_DevM := "STATUS_450"."UC21-TA03".Main, XS_Parameter := "HMI_PARAM_450"."GL03-MA01", XS_Command := "HMI_CMD_450"."GL03-MA01", OS_Status => "STATUS_450"."GL03-MA01", OB1OutDir1 => #TS_UC21TA03.ReqDir1, OB1OutDir2 => #TS_UC21TA03.ReqDir2)
   END_RUNG
   // the same network as SCL:
   #SF_GL03_MA01(IS_ZoneM := "STATUS_Zone400".Station450_Mode.Main,   // "STD_Drive1"
                 IS_ZoneS := "STATUS_Zone400".Station450_Mode.Specific,
                 IB1GenRelDir1 := #TS_GL03MA01.GenRelDir1,
                 IB1GenRelDir2 := #TS_GL03MA01.GenRelDir2,
                 IB1IntlDir1 := #TS_GL03MA01.IntlDir1,
                 IB1IntlDir2 := #TS_GL03MA01.IntlDir2,
                 IB1AutDir1 := #TS_GL03MA01.AutDir1,
                 IB1AutDir2 := #TS_GL03MA01.AutDir2,
                 IB1DevFdbDir1 := "STATUS_450"."UC21-TA03".Specific.OutDir1,
                 IB1DevFdbDir2 := "STATUS_450"."UC21-TA03".Specific.OutDir2,
                 IB1AlmSupp := "STATUS_Zone400".Station450_Mode.Specific.AlmSupp,
                 IB1ManDir1 := #TS_GL03MA01.ManDir1,
                 IB1ManDir2 := #TS_GL03MA01.ManDir2,
                 IS_DevM := "STATUS_450"."UC21-TA03".Main,
                 XS_Parameter := "HMI_PARAM_450"."GL03-MA01",
                 XS_Command := "HMI_CMD_450"."GL03-MA01",
                 OS_Status => "STATUS_450"."GL03-MA01",
                 OB1OutDir1 => #TS_UC21TA03.ReqDir1,
                 OB1OutDir2 => #TS_UC21TA03.ReqDir2);
END_REGION

REGION Network 41: UC21_TA03 - Speed setpoint
   RUNG wire#powerrail
      Move(in := "ProdParam"."450_GL03_ConvSpeedSlow", out1 => #TS_UC21TA03.SpeedSP)
   END_RUNG
   RUNG wire#powerrail
      I_Contact( "STATUS_Zone400".Station450_Mode.Main.Man )
      Move(in := "ProdParam"."450_GL03_ConvSpeed", out1 => #TS_UC21TA03.SpeedSP)
   END_RUNG
   // the same network as SCL:
   #TS_UC21TA03.SpeedSP := "ProdParam"."450_GL03_ConvSpeedSlow";
   IF NOT "STATUS_Zone400".Station450_Mode.Main.Man THEN
       #TS_UC21TA03.SpeedSP := "ProdParam"."450_GL03_ConvSpeed";
   END_IF;
END_REGION

REGION Network 42: UC21_TA03 - Frequency convertor block call
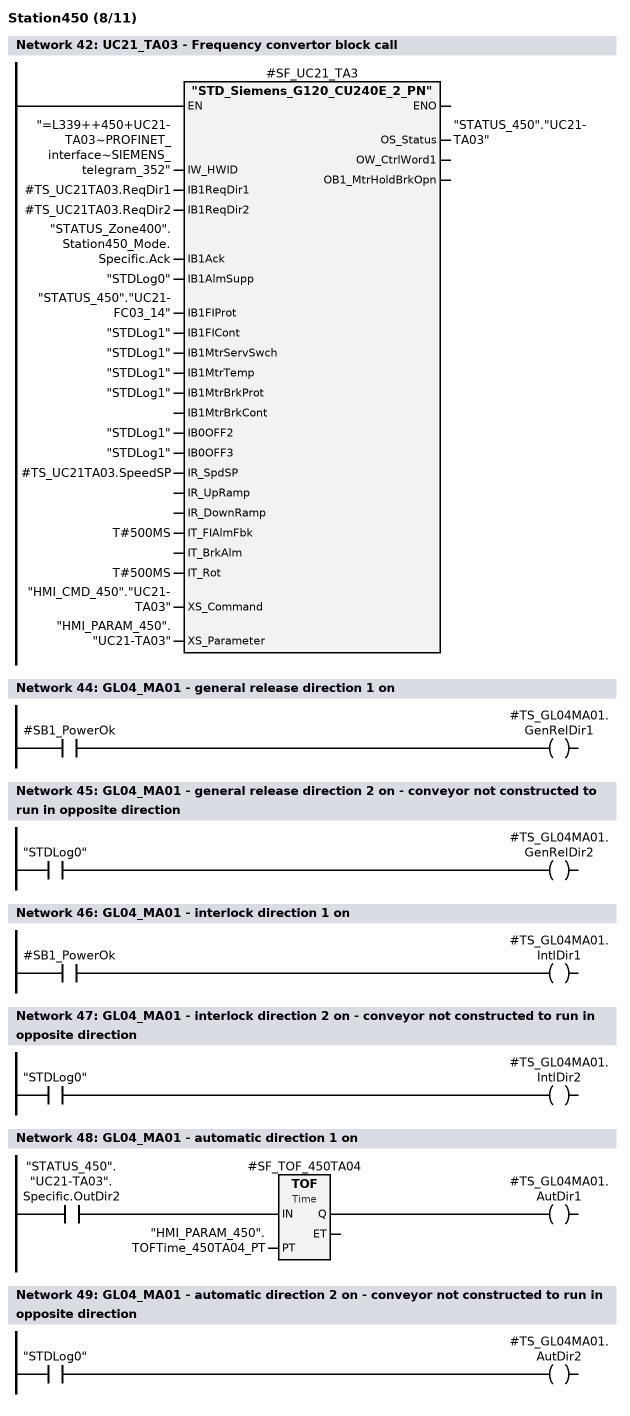
   RUNG wire#powerrail
      #SF_UC21_TA3(IW_HWID := "=L339++450+UC21-TA03~PROFINET_interface~SIEMENS_telegram_352", IB1ReqDir1 := #TS_UC21TA03.ReqDir1, IB1ReqDir2 := #TS_UC21TA03.ReqDir2, IB1Ack := "STATUS_Zone400".Station450_Mode.Specific.Ack, IB1AlmSupp := "STDLog0", IB1FIProt := "STATUS_450"."UC21-FC03_14", IB1FICont := "STDLog1", IB1MtrServSwch := "STDLog1", IB1MtrTemp := "STDLog1", IB1MtrBrkProt := "STDLog1", IB1MtrBrkCont :=, IB0OFF2 := "STDLog1", IB0OFF3 := "STDLog1", IR_SpdSP := #TS_UC21TA03.SpeedSP, IR_UpRamp :=, IR_DownRamp :=, IT_FIAlmFbk := T#500MS, IT_BrkAlm :=, IT_Rot := T#500MS, XS_Command := "HMI_CMD_450"."UC21-TA03", XS_Parameter := "HMI_PARAM_450"."UC21-TA03", OS_Status => "STATUS_450"."UC21-TA03", OW_CtrlWord1 =>, OB1_MtrHoldBrkOpn =>)
   END_RUNG
   // the same network as SCL:
   #SF_UC21_TA3(IW_HWID := "=L339++450+UC21-TA03~PROFINET_interface~SIEMENS_telegram_352",   // "STD_Siemens_G120_CU240E_2_PN"
                IB1ReqDir1 := #TS_UC21TA03.ReqDir1,
                IB1ReqDir2 := #TS_UC21TA03.ReqDir2,
                IB1Ack := "STATUS_Zone400".Station450_Mode.Specific.Ack,
                IB1AlmSupp := "STDLog0",
                IB1FIProt := "STATUS_450"."UC21-FC03_14",
                IB1FICont := "STDLog1",
                IB1MtrServSwch := "STDLog1",
                IB1MtrTemp := "STDLog1",
                IB1MtrBrkProt := "STDLog1",
                IB0OFF2 := "STDLog1",
                IB0OFF3 := "STDLog1",
                IR_SpdSP := #TS_UC21TA03.SpeedSP,
                IT_FIAlmFbk := T#500MS,
                IT_Rot := T#500MS,
                XS_Command := "HMI_CMD_450"."UC21-TA03",
                XS_Parameter := "HMI_PARAM_450"."UC21-TA03",
                OS_Status => "STATUS_450"."UC21-TA03");
END_REGION

REGION Network 43: ***************GL04_MA01 Conveyor M6***************
END_REGION

REGION Network 44: GL04_MA01 - general release direction 1 on
   RUNG wire#powerrail
      Contact( #SB1_PowerOk )
      Coil( #TS_GL04MA01.GenRelDir1 )
   END_RUNG
   // the same network as SCL:
   #TS_GL04MA01.GenRelDir1 := #SB1_PowerOk;
END_REGION

REGION Network 45: GL04_MA01 - general release direction 2 on - conveyor not constructed to run in opposite direction
   RUNG wire#powerrail
      Contact( "STDLog0" )
      Coil( #TS_GL04MA01.GenRelDir2 )
   END_RUNG
   // the same network as SCL:
   #TS_GL04MA01.GenRelDir2 := "STDLog0";
END_REGION

REGION Network 46: GL04_MA01 - interlock direction 1 on
   RUNG wire#powerrail
      Contact( #SB1_PowerOk )
      Coil( #TS_GL04MA01.IntlDir1 )
   END_RUNG
   // the same network as SCL:
   #TS_GL04MA01.IntlDir1 := #SB1_PowerOk;
END_REGION

REGION Network 47: GL04_MA01 - interlock direction 2 on - conveyor not constructed to run in opposite direction
   RUNG wire#powerrail
      Contact( "STDLog0" )
      Coil( #TS_GL04MA01.IntlDir2 )
   END_RUNG
   // the same network as SCL:
   #TS_GL04MA01.IntlDir2 := "STDLog0";
END_REGION

REGION Network 48: GL04_MA01 - automatic direction 1 on
   RUNG wire#powerrail
      Contact( "STATUS_450"."UC21-TA03".Specific.OutDir2 )
      { S7_Templates := "time_type := Time" } #SF_TOF_450TA04.TOF(pt := "HMI_PARAM_450".TOFTime_450TA04_PT, et =>)
      Coil( #TS_GL04MA01.AutDir1 )
   END_RUNG
   // the same network as SCL:
   #SF_TOF_450TA04(IN := "STATUS_450"."UC21-TA03".Specific.OutDir2, PT := "HMI_PARAM_450".TOFTime_450TA04_PT);   // TOF
   #TS_GL04MA01.AutDir1 := #SF_TOF_450TA04.Q;
END_REGION

REGION Network 49: GL04_MA01 - automatic direction 2 on - conveyor not constructed to run in opposite direction
   RUNG wire#powerrail
      Contact( "STDLog0" )
      Coil( #TS_GL04MA01.AutDir2 )
   END_RUNG
   // the same network as SCL:
   #TS_GL04MA01.AutDir2 := "STDLog0";
END_REGION

REGION Network 50: GL04_MA01 - manual direction 1 on
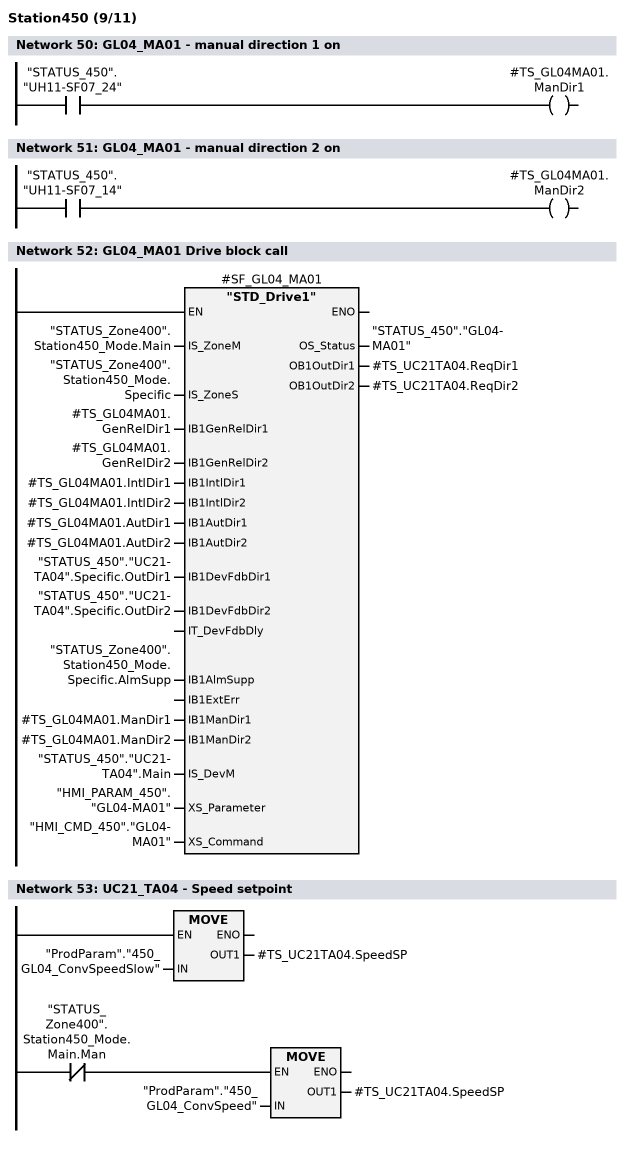
   RUNG wire#powerrail
      Contact( "STATUS_450"."UH11-SF07_24" )
      Coil( #TS_GL04MA01.ManDir1 )
   END_RUNG
   // the same network as SCL:
   #TS_GL04MA01.ManDir1 := "STATUS_450"."UH11-SF07_24";
END_REGION

REGION Network 51: GL04_MA01 - manual direction 2 on
   RUNG wire#powerrail
      Contact( "STATUS_450"."UH11-SF07_14" )
      Coil( #TS_GL04MA01.ManDir2 )
   END_RUNG
   // the same network as SCL:
   #TS_GL04MA01.ManDir2 := "STATUS_450"."UH11-SF07_14";
END_REGION

REGION Network 52: GL04_MA01 Drive block call
   RUNG wire#powerrail
      #SF_GL04_MA01(IS_ZoneM := "STATUS_Zone400".Station450_Mode.Main, IS_ZoneS := "STATUS_Zone400".Station450_Mode.Specific, IB1GenRelDir1 := #TS_GL04MA01.GenRelDir1, IB1GenRelDir2 := #TS_GL04MA01.GenRelDir2, IB1IntlDir1 := #TS_GL04MA01.IntlDir1, IB1IntlDir2 := #TS_GL04MA01.IntlDir2, IB1AutDir1 := #TS_GL04MA01.AutDir1, IB1AutDir2 := #TS_GL04MA01.AutDir2, IB1DevFdbDir1 := "STATUS_450"."UC21-TA04".Specific.OutDir1, IB1DevFdbDir2 := "STATUS_450"."UC21-TA04".Specific.OutDir2, IT_DevFdbDly :=, IB1AlmSupp := "STATUS_Zone400".Station450_Mode.Specific.AlmSupp, IB1ExtErr :=, IB1ManDir1 := #TS_GL04MA01.ManDir1, IB1ManDir2 := #TS_GL04MA01.ManDir2, IS_DevM := "STATUS_450"."UC21-TA04".Main, XS_Parameter := "HMI_PARAM_450"."GL04-MA01", XS_Command := "HMI_CMD_450"."GL04-MA01", OS_Status => "STATUS_450"."GL04-MA01", OB1OutDir1 => #TS_UC21TA04.ReqDir1, OB1OutDir2 => #TS_UC21TA04.ReqDir2)
   END_RUNG
   // the same network as SCL:
   #SF_GL04_MA01(IS_ZoneM := "STATUS_Zone400".Station450_Mode.Main,   // "STD_Drive1"
                 IS_ZoneS := "STATUS_Zone400".Station450_Mode.Specific,
                 IB1GenRelDir1 := #TS_GL04MA01.GenRelDir1,
                 IB1GenRelDir2 := #TS_GL04MA01.GenRelDir2,
                 IB1IntlDir1 := #TS_GL04MA01.IntlDir1,
                 IB1IntlDir2 := #TS_GL04MA01.IntlDir2,
                 IB1AutDir1 := #TS_GL04MA01.AutDir1,
                 IB1AutDir2 := #TS_GL04MA01.AutDir2,
                 IB1DevFdbDir1 := "STATUS_450"."UC21-TA04".Specific.OutDir1,
                 IB1DevFdbDir2 := "STATUS_450"."UC21-TA04".Specific.OutDir2,
                 IB1AlmSupp := "STATUS_Zone400".Station450_Mode.Specific.AlmSupp,
                 IB1ManDir1 := #TS_GL04MA01.ManDir1,
                 IB1ManDir2 := #TS_GL04MA01.ManDir2,
                 IS_DevM := "STATUS_450"."UC21-TA04".Main,
                 XS_Parameter := "HMI_PARAM_450"."GL04-MA01",
                 XS_Command := "HMI_CMD_450"."GL04-MA01",
                 OS_Status => "STATUS_450"."GL04-MA01",
                 OB1OutDir1 => #TS_UC21TA04.ReqDir1,
                 OB1OutDir2 => #TS_UC21TA04.ReqDir2);
END_REGION

REGION Network 53: UC21_TA04 - Speed setpoint
   RUNG wire#powerrail
      Move(in := "ProdParam"."450_GL04_ConvSpeedSlow", out1 => #TS_UC21TA04.SpeedSP)
   END_RUNG
   RUNG wire#powerrail
      I_Contact( "STATUS_Zone400".Station450_Mode.Main.Man )
      Move(in := "ProdParam"."450_GL04_ConvSpeed", out1 => #TS_UC21TA04.SpeedSP)
   END_RUNG
   // the same network as SCL:
   #TS_UC21TA04.SpeedSP := "ProdParam"."450_GL04_ConvSpeedSlow";
   IF NOT "STATUS_Zone400".Station450_Mode.Main.Man THEN
       #TS_UC21TA04.SpeedSP := "ProdParam"."450_GL04_ConvSpeed";
   END_IF;
END_REGION

REGION Network 54: UC21_TA04 - Frequency convertor block call
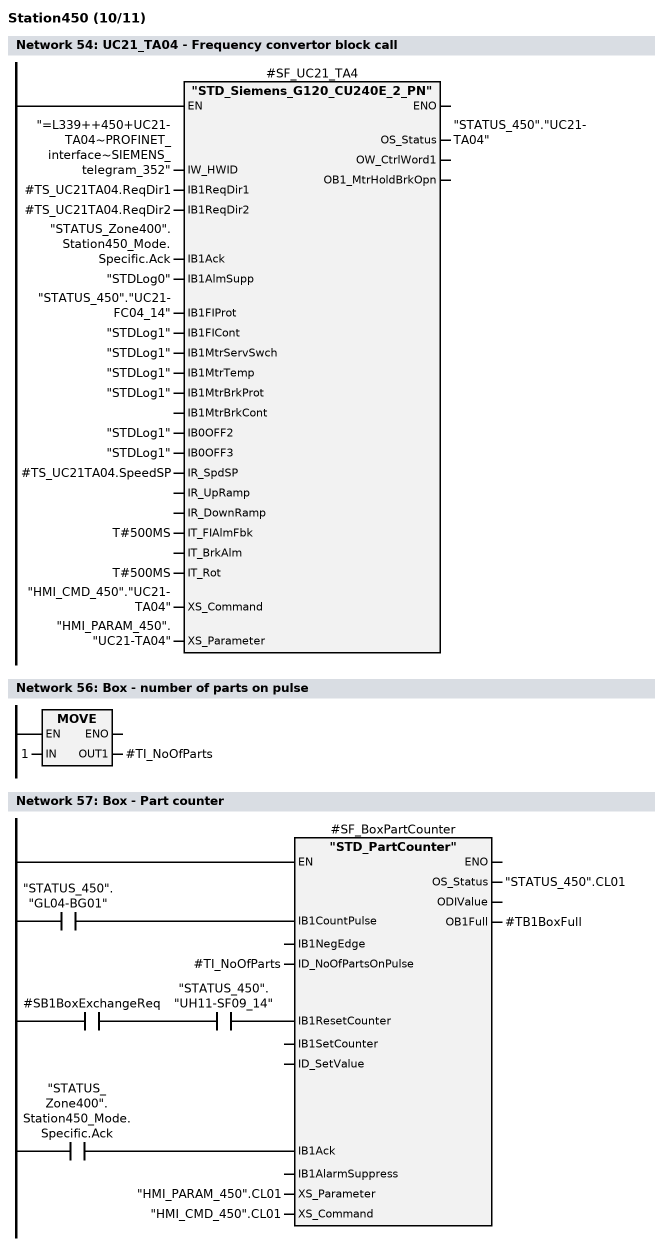
   RUNG wire#powerrail
      #SF_UC21_TA4(IW_HWID := "=L339++450+UC21-TA04~PROFINET_interface~SIEMENS_telegram_352", IB1ReqDir1 := #TS_UC21TA04.ReqDir1, IB1ReqDir2 := #TS_UC21TA04.ReqDir2, IB1Ack := "STATUS_Zone400".Station450_Mode.Specific.Ack, IB1AlmSupp := "STDLog0", IB1FIProt := "STATUS_450"."UC21-FC04_14", IB1FICont := "STDLog1", IB1MtrServSwch := "STDLog1", IB1MtrTemp := "STDLog1", IB1MtrBrkProt := "STDLog1", IB1MtrBrkCont :=, IB0OFF2 := "STDLog1", IB0OFF3 := "STDLog1", IR_SpdSP := #TS_UC21TA04.SpeedSP, IR_UpRamp :=, IR_DownRamp :=, IT_FIAlmFbk := T#500MS, IT_BrkAlm :=, IT_Rot := T#500MS, XS_Command := "HMI_CMD_450"."UC21-TA04", XS_Parameter := "HMI_PARAM_450"."UC21-TA04", OS_Status => "STATUS_450"."UC21-TA04", OW_CtrlWord1 =>, OB1_MtrHoldBrkOpn =>)
   END_RUNG
   // the same network as SCL:
   #SF_UC21_TA4(IW_HWID := "=L339++450+UC21-TA04~PROFINET_interface~SIEMENS_telegram_352",   // "STD_Siemens_G120_CU240E_2_PN"
                IB1ReqDir1 := #TS_UC21TA04.ReqDir1,
                IB1ReqDir2 := #TS_UC21TA04.ReqDir2,
                IB1Ack := "STATUS_Zone400".Station450_Mode.Specific.Ack,
                IB1AlmSupp := "STDLog0",
                IB1FIProt := "STATUS_450"."UC21-FC04_14",
                IB1FICont := "STDLog1",
                IB1MtrServSwch := "STDLog1",
                IB1MtrTemp := "STDLog1",
                IB1MtrBrkProt := "STDLog1",
                IB0OFF2 := "STDLog1",
                IB0OFF3 := "STDLog1",
                IR_SpdSP := #TS_UC21TA04.SpeedSP,
                IT_FIAlmFbk := T#500MS,
                IT_Rot := T#500MS,
                XS_Command := "HMI_CMD_450"."UC21-TA04",
                XS_Parameter := "HMI_PARAM_450"."UC21-TA04",
                OS_Status => "STATUS_450"."UC21-TA04");
END_REGION

REGION Network 55: *************** Box ***************
END_REGION

REGION Network 56: Box - number of parts on pulse
   RUNG wire#powerrail
      Move(in := 1, out1 => #TI_NoOfParts)
   END_RUNG
   // the same network as SCL:
   #TI_NoOfParts := 1;
END_REGION

REGION Network 57: Box - Part counter
   RUNG wire#powerrail
      #SF_BoxPartCounter(IB1CountPulse := wire#w1, IB1ResetCounter := wire#w2, IB1Ack := wire#w3, IB1NegEdge :=, ID_NoOfPartsOnPulse := #TI_NoOfParts, IB1SetCounter :=, ID_SetValue :=, IB1AlarmSuppress :=, XS_Parameter := "HMI_PARAM_450".CL01, XS_Command := "HMI_CMD_450".CL01, OS_Status => "STATUS_450".CL01, ODIValue =>, OB1Full => #TB1BoxFull)
   END_RUNG
   RUNG wire#powerrail
      Contact( "STATUS_450"."GL04-BG01" )
   END_RUNG wire#w1
   RUNG wire#powerrail
      Contact( #SB1BoxExchangeReq )
      Contact( "STATUS_450"."UH11-SF09_14" )
   END_RUNG wire#w2
   RUNG wire#powerrail
      Contact( "STATUS_Zone400".Station450_Mode.Specific.Ack )
   END_RUNG wire#w3
   // the same network as SCL:
   #SF_BoxPartCounter(IB1CountPulse := "STATUS_450"."GL04-BG01",   // "STD_PartCounter"
                      ID_NoOfPartsOnPulse := #TI_NoOfParts,
                      IB1ResetCounter := #SB1BoxExchangeReq AND "STATUS_450"."UH11-SF09_14",
                      IB1Ack := "STATUS_Zone400".Station450_Mode.Specific.Ack,
                      XS_Parameter := "HMI_PARAM_450".CL01,
                      XS_Command := "HMI_CMD_450".CL01,
                      OS_Status => "STATUS_450".CL01,
                      OB1Full => #TB1BoxFull);
END_REGION

REGION Network 58: Box - exchange request
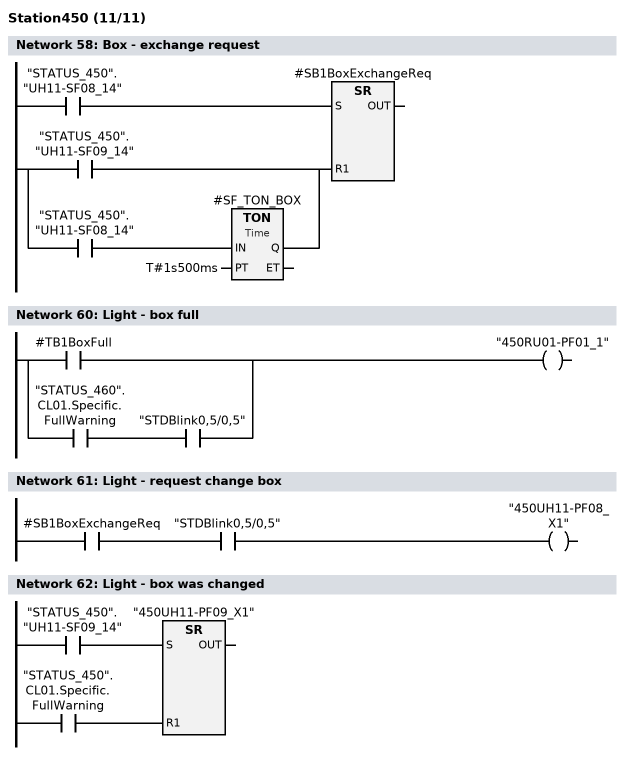
   RUNG wire#powerrail
      Contact( "STATUS_450"."UH11-SF08_14" )
      S_SR(operand := #SB1BoxExchangeReq, r1 := wire#w1)
   END_RUNG
   RUNG wire#powerrail
      Contact( "STATUS_450"."UH11-SF09_14" )
   END_RUNG wire#w1
   RUNG wire#powerrail
      Contact( "STATUS_450"."UH11-SF08_14" )
      { S7_Templates := "time_type := Time" } #SF_TON_BOX.TON(pt := T#1s500ms, et =>)
   END_RUNG wire#w1
   // the same network as SCL:
   #SF_TON_BOX(IN := "STATUS_450"."UH11-SF08_14", PT := T#1s500ms);   // TON
   IF "STATUS_450"."UH11-SF08_14" THEN
       #SB1BoxExchangeReq := TRUE;   // SR flip-flop
   END_IF;
   IF "STATUS_450"."UH11-SF09_14" OR #SF_TON_BOX.Q THEN #SB1BoxExchangeReq := FALSE; END_IF;
END_REGION

REGION Network 59: *************** Signalization ***************
END_REGION

REGION Network 60: Light - box full
   RUNG wire#powerrail
      Contact( #TB1BoxFull )
      wire#w1
      Coil( "450RU01-PF01_1" )
   END_RUNG
   RUNG wire#powerrail
      Contact( "STATUS_460".CL01.Specific.FullWarning )
      Contact( "STDBlink0,5/0,5" )
   END_RUNG wire#w1
   // the same network as SCL:
   "450RU01-PF01_1" := #TB1BoxFull OR ("STATUS_460".CL01.Specific.FullWarning AND "STDBlink0,5/0,5");
END_REGION

REGION Network 61: Light - request change box
   RUNG wire#powerrail
      Contact( #SB1BoxExchangeReq )
      Contact( "STDBlink0,5/0,5" )
      Coil( "450UH11-PF08_X1" )
   END_RUNG
   // the same network as SCL:
   "450UH11-PF08_X1" := #SB1BoxExchangeReq AND "STDBlink0,5/0,5";
END_REGION

REGION Network 62: Light - box was changed
   RUNG wire#powerrail
      Contact( "STATUS_450"."UH11-SF09_14" )
      S_SR(operand := "450UH11-PF09_X1", r1 := wire#w1)
   END_RUNG
   RUNG wire#powerrail
      Contact( "STATUS_450".CL01.Specific.FullWarning )
   END_RUNG wire#w1
   // the same network as SCL:
   IF "STATUS_450"."UH11-SF09_14" THEN
       "450UH11-PF09_X1" := TRUE;   // SR flip-flop
   END_IF;
   IF "STATUS_450".CL01.Specific.FullWarning THEN "450UH11-PF09_X1" := FALSE; END_IF;
END_REGION
END_FUNCTION_BLOCK
